// TIA Portal V18 export
// export: Created 2026-01-09T11:31:52.0930933Z, ExportSetting WithDefaults, DisplayName Totally Integrated Automation Portal, DisplayVersion V18 Update 5, DisplayName TIA Portal Openness, DisplayVersion V18 Update 5, DisplayName TIA Portal Teamcenter Gateway, DisplayVersion V18, DisplayName TIA Portal Version Control Interface, DisplayVersion V18, DisplayName SINAMICS Startdrive Advanced, DisplayVersion V18 SP2 Update 1, DisplayName SINAMICS Startdrive G110M, G120, G120C, G120D, G120P, G115D, DisplayVersion V18 SP2 Update 1, DisplayName SINAMICS Startdrive G130, G150, S120, S150, SINAMICS MV, S210, G220, S200, DisplayVersion V18 SP2 Update 1, DisplayName STEP 7 Professional, DisplayVersion V18 Update 5, DisplayName STEP 7 Safety, DisplayVersion V18, DisplayName WinCC Professional, DisplayVersion V18 Update 5
TagTable "ChangeOverProcess"
  AutoProcessData_A_Table_1{1}_PartStatus : Int  (PLC tag AutoProcessData.A_Table_1[1].PartStatus, CPU S71500-2PN_TP700, 1 s)
  AutoProcessData_A_Table_1{2}_PartStatus : Int  (PLC tag AutoProcessData.A_Table_1[2].PartStatus, CPU S71500-2PN_TP700, 1 s)
  AutoProcessData_A_Table_1{3}_PartStatus : Int  (PLC tag AutoProcessData.A_Table_1[3].PartStatus, CPU S71500-2PN_TP700, 1 s)
  AutoProcessData_A_Table_1{4}_PartStatus : Int  (PLC tag AutoProcessData.A_Table_1[4].PartStatus, CPU S71500-2PN_TP700, 1 s)
  AutoProcessData_A_Table_1{5}_PartStatus : Int  (PLC tag AutoProcessData.A_Table_1[5].PartStatus, CPU S71500-2PN_TP700, 1 s)
  AutoProcessData_A_Table_1{6}_PartStatus : Int  (PLC tag AutoProcessData.A_Table_1[6].PartStatus, CPU S71500-2PN_TP700, 1 s)
  AutoProcessData_A_Table_1{7}_PartStatus : Int  (PLC tag AutoProcessData.A_Table_1[7].PartStatus, CPU S71500-2PN_TP700, 1 s)
  AutoProcessData_A_Table_1{8}_PartStatus : Int  (PLC tag AutoProcessData.A_Table_1[8].PartStatus, CPU S71500-2PN_TP700, 1 s)
  AutoProcessData_A_Table_2{1}_PartStatus : Int  (PLC tag AutoProcessData.A_Table_2[1].PartStatus, CPU S71500-2PN_TP700, 1 s)
  AutoProcessData_A_Table_2{2}_PartStatus : Int  (PLC tag AutoProcessData.A_Table_2[2].PartStatus, CPU S71500-2PN_TP700, 1 s)
  AutoProcessData_A_Table_2{3}_PartStatus : Int  (PLC tag AutoProcessData.A_Table_2[3].PartStatus, CPU S71500-2PN_TP700, 1 s)
  AutoProcessData_A_Table_2{4}_PartStatus : Int  (PLC tag AutoProcessData.A_Table_2[4].PartStatus, CPU S71500-2PN_TP700, 1 s)
  AutoProcessData_A_Table_2{5}_PartStatus : Int  (PLC tag AutoProcessData.A_Table_2[5].PartStatus, CPU S71500-2PN_TP700, 1 s)
  AutoProcessData_A_Table_2{6}_PartStatus : Int  (PLC tag AutoProcessData.A_Table_2[6].PartStatus, CPU S71500-2PN_TP700, 1 s)
  AutoProcessData_A_Table_2{7}_PartStatus : Int  (PLC tag AutoProcessData.A_Table_2[7].PartStatus, CPU S71500-2PN_TP700, 1 s)
  AutoProcessData_A_Table_2{8}_PartStatus : Int  (PLC tag AutoProcessData.A_Table_2[8].PartStatus, CPU S71500-2PN_TP700, 1 s)
  AutoProcessData_GlobalData_Table1CodeOKFlag : Bool  (PLC tag AutoProcessData.GlobalData.Table1CodeOKFlag, CPU S71500-2PN_TP700, 1 s)
  AutoProcessData_GlobalData_Table2CodeOKFlag : Bool  (PLC tag AutoProcessData.GlobalData.Table2CodeOKFlag, CPU S71500-2PN_TP700, 1 s)
  AutoProcessData_GlobalData_Fixture1CodeOKFlag : Bool  (PLC tag AutoProcessData.GlobalData.Fixture1CodeOKFlag, CPU S71500-2PN_TP700, 1 s)
  AutoProcessData_GlobalData_Fixture2CodeOKFlag : Bool  (PLC tag AutoProcessData.GlobalData.Fixture2CodeOKFlag, CPU S71500-2PN_TP700, 1 s)
  AutoProcessData_GlobalData_Robot2GripperCodeOKFlag : Bool  (PLC tag AutoProcessData.GlobalData.Robot2GripperCodeOKFlag, CPU S71500-2PN_TP700, 1 s)
  AutoProcessData_GlobalData_Robot1GripperCodeOKFlag : Bool  (PLC tag AutoProcessData.GlobalData.Robot1GripperCodeOKFlag, CPU S71500-2PN_TP700, 1 s)
  AutoProcessData_GlobalData_Robot3GripperCodeOKFlag : Bool  (PLC tag AutoProcessData.GlobalData.Robot3GripperCodeOKFlag, CPU S71500-2PN_TP700, 1 s)
  AutoProcessData_GlobalData_Robot1GripCodeStatus1 : Int  (PLC tag AutoProcessData.GlobalData.Robot1GripCodeStatus1, CPU S71500-2PN_TP700, 1 s)
  AutoProcessData_GlobalData_Robot1GripCodeStatus2 : Int  (PLC tag AutoProcessData.GlobalData.Robot1GripCodeStatus2, CPU S71500-2PN_TP700, 1 s)
  AutoProcessData_GlobalData_Robot1GripCodeStatus3 : Int  (PLC tag AutoProcessData.GlobalData.Robot1GripCodeStatus3, CPU S71500-2PN_TP700, 1 s)
  AutoProcessData_GlobalData_Robot1GripCodeStatus4 : Int  (PLC tag AutoProcessData.GlobalData.Robot1GripCodeStatus4, CPU S71500-2PN_TP700, 1 s)
  AutoProcessData_GlobalData_Robot2GripCodeStatus1 : Int  (PLC tag AutoProcessData.GlobalData.Robot2GripCodeStatus1, CPU S71500-2PN_TP700, 1 s)
  AutoProcessData_GlobalData_Robot2GripCodeStatus2 : Int  (PLC tag AutoProcessData.GlobalData.Robot2GripCodeStatus2, CPU S71500-2PN_TP700, 1 s)
  AutoProcessData_GlobalData_Robot2GripCodeStatus3 : Int  (PLC tag AutoProcessData.GlobalData.Robot2GripCodeStatus3, CPU S71500-2PN_TP700, 1 s)
  AutoProcessData_GlobalData_Robot2GripCodeStatus4 : Int  (PLC tag AutoProcessData.GlobalData.Robot2GripCodeStatus4, CPU S71500-2PN_TP700, 1 s)
  AutoProcessData_GlobalData_Robot3GripCodeStatus1 : Int  (PLC tag AutoProcessData.GlobalData.Robot3GripCodeStatus1, CPU S71500-2PN_TP700, 1 s)
  AutoProcessData_GlobalData_Robot3GripCodeStatus2 : Int  (PLC tag AutoProcessData.GlobalData.Robot3GripCodeStatus2, CPU S71500-2PN_TP700, 1 s)
  AutoProcessData_GlobalData_Robot3GripCodeStatus3 : Int  (PLC tag AutoProcessData.GlobalData.Robot3GripCodeStatus3, CPU S71500-2PN_TP700, 1 s)
  AutoProcessData_GlobalData_Robot3GripCodeStatus4 : Int  (PLC tag AutoProcessData.GlobalData.Robot3GripCodeStatus4, CPU S71500-2PN_TP700, 1 s)
  AutoProcessData_GlobalData_FixtureCode_A1Status1 : Int  (PLC tag AutoProcessData.GlobalData.FixtureCode_A1Status1, CPU S71500-2PN_TP700, 1 s)
  AutoProcessData_GlobalData_FixtureCode_A1Status2 : Int  (PLC tag AutoProcessData.GlobalData.FixtureCode_A1Status2, CPU S71500-2PN_TP700, 1 s)
  AutoProcessData_GlobalData_FixtureCode_A1Status3 : Int  (PLC tag AutoProcessData.GlobalData.FixtureCode_A1Status3, CPU S71500-2PN_TP700, 1 s)
  AutoProcessData_GlobalData_FixtureCode_A1Status4 : Int  (PLC tag AutoProcessData.GlobalData.FixtureCode_A1Status4, CPU S71500-2PN_TP700, 1 s)
  AutoProcessData_GlobalData_FixtureCode_A1Status5 : Int  (PLC tag AutoProcessData.GlobalData.FixtureCode_A1Status5, CPU S71500-2PN_TP700, 1 s)
  AutoProcessData_GlobalData_FixtureCode_A1Status6 : Int  (PLC tag AutoProcessData.GlobalData.FixtureCode_A1Status6, CPU S71500-2PN_TP700, 1 s)
  AutoProcessData_GlobalData_FixtureCode_A1Status7 : Int  (PLC tag AutoProcessData.GlobalData.FixtureCode_A1Status7, CPU S71500-2PN_TP700, 1 s)
  AutoProcessData_GlobalData_FixtureCode_A1Status8 : Int  (PLC tag AutoProcessData.GlobalData.FixtureCode_A1Status8, CPU S71500-2PN_TP700, 1 s)
  AutoProcessData_GlobalData_FixtureCode_A1Status9 : Int  (PLC tag AutoProcessData.GlobalData.FixtureCode_A1Status9, CPU S71500-2PN_TP700, 1 s)
  AutoProcessData_GlobalData_FixtureCode_A1Status10 : Int  (PLC tag AutoProcessData.GlobalData.FixtureCode_A1Status10, CPU S71500-2PN_TP700, 1 s)
  AutoProcessData_GlobalData_FixtureCode_A2Status1 : Int  (PLC tag AutoProcessData.GlobalData.FixtureCode_A2Status1, CPU S71500-2PN_TP700, 1 s)
  AutoProcessData_GlobalData_FixtureCode_A2Status2 : Int  (PLC tag AutoProcessData.GlobalData.FixtureCode_A2Status2, CPU S71500-2PN_TP700, 1 s)
  AutoProcessData_GlobalData_FixtureCode_A2Status3 : Int  (PLC tag AutoProcessData.GlobalData.FixtureCode_A2Status3, CPU S71500-2PN_TP700, 1 s)
  AutoProcessData_GlobalData_FixtureCode_A2Status4 : Int  (PLC tag AutoProcessData.GlobalData.FixtureCode_A2Status4, CPU S71500-2PN_TP700, 1 s)
  AutoProcessData_GlobalData_FixtureCode_A2Status5 : Int  (PLC tag AutoProcessData.GlobalData.FixtureCode_A2Status5, CPU S71500-2PN_TP700, 1 s)
  AutoProcessData_GlobalData_FixtureCode_A2Status6 : Int  (PLC tag AutoProcessData.GlobalData.FixtureCode_A2Status6, CPU S71500-2PN_TP700, 1 s)
  AutoProcessData_GlobalData_FixtureCode_A2Status7 : Int  (PLC tag AutoProcessData.GlobalData.FixtureCode_A2Status7, CPU S71500-2PN_TP700, 1 s)
  AutoProcessData_GlobalData_FixtureCode_A2Status8 : Int  (PLC tag AutoProcessData.GlobalData.FixtureCode_A2Status8, CPU S71500-2PN_TP700, 1 s)
  AutoProcessData_GlobalData_FixtureCode_A2Status9 : Int  (PLC tag AutoProcessData.GlobalData.FixtureCode_A2Status9, CPU S71500-2PN_TP700, 1 s)
  AutoProcessData_GlobalData_FixtureCode_A2Status10 : Int  (PLC tag AutoProcessData.GlobalData.FixtureCode_A2Status10, CPU S71500-2PN_TP700, 1 s)
  ChangeOver_DB_Global_ChangeOverFinish : Bool  (PLC tag ChangeOver_DB.Global.AllFixtureScanCompareOk, CPU S71500-2PN_TP700, 1 s)
  ChangeOver_DB_Global_ChangeOverRequest : Bool  (PLC tag ChangeOver_DB.Global.ChangeOverRequest, CPU S71500-2PN_TP700, 1 s)
  ChangeOver_DB_Global_Hmi_Confirm_ChangeOver : Bool  (PLC tag ChangeOver_DB.Global.Hmi_Confirm_ChangeOver, CPU S71500-2PN_TP700, 1 s)
  ChangeOver_DB_Global_ScanFixtureFlag : Bool  (PLC tag ChangeOver_DB.Global.ScanFixtureFlag, CPU S71500-2PN_TP700, 1 s)
  ChangeOver_DB_Global_ChangeOverSelected : Bool  (PLC tag ChangeOver_DB.Global.ChangeOverSelected, CPU S71500-2PN_TP700, 1 s)
